// TIA Portal project "PLC_test_DATN" (V16)

(* hardware
DEVICE "S7-1200 station_1"  S7-1200 Station
   slot 0: "Rack_0"  S7-1200 Rack  Rack  V1.0
   slot 1: "PLC_2"  CPU 1214C DC/DC/DC  6ES7 214-1AG40-0XB0  V4.4
*)

// ===== PLC "PLC_2"  CPU 1214C DC/DC/DC =====

VAR_GLOBAL   // PLC tag table "Default tag table"
   "START BUTTON" AT %I0.0 : Bool;
   "SSBELTBEGIN" AT %I0.1 : Bool;
   "SSZ+" AT %I1.3 : Bool;
   "SSZ-" AT %I1.4 : Bool;
   "STOP BUTTON" AT %I1.5 : Bool;
   "GRAB" AT %I1.6 : Bool;
   "LETOUT" AT %I1.7 : Bool;
   "SSX0" AT %I1.0 : Bool;
   "SSX1" AT %I1.1 : Bool;
   "SSX2" AT %I0.4 : Bool;
   "Tag_2" AT %I0.5 : Bool;
   "Tag_3" AT %I0.6 : Bool;
   "SSBELTEND" AT %I0.7 : Bool;
   "SSPUSHERBACK" AT %I0.2 : Bool;
   "SSX3" AT %I1.2 : Bool;
   "SSPUSHERFRONT" AT %I0.3 : Bool;
   "BELTMOTOR" AT %Q0.0 : Bool;
   "HANDPICK" AT %Q0.1 : Bool;
   "HANDLEFT" AT %Q0.3 : Bool;
   "HANDUP" AT %Q0.2 : Bool;
   "PUSHERFRONT" AT %Q0.4 : Bool;
   "HANDRELEASE" AT %Q0.5 : Bool;
   "PUSHERBACK" AT %Q1.1 : Bool;
   "ZPLUS" AT %Q1.2 : Bool;
   "ZMINUS" AT %Q1.3 : Bool;
   "G" AT %Q1.4 : Bool;
   "HANDDOWN" AT %Q0.6 : Bool;
   "HANDRIGHT" AT %Q0.7 : Bool;
   "Tag_12" AT %Q1.0 : Bool;
   "System_Byte" AT %MB2000 : Byte;
   "FirstScan" AT %M2000.0 : Bool;
   "DiagStatusUpdate" AT %M2000.1 : Bool;
   "AlwaysTRUE" AT %M2000.2 : Bool;
   "AlwaysFALSE" AT %M2000.3 : Bool;
   "Clock_Byte" AT %MB5000 : Byte;
   "Clock_10Hz" AT %M5000.0 : Bool;
   "Clock_5Hz" AT %M5000.1 : Bool;
   "Clock_2.5Hz" AT %M5000.2 : Bool;
   "Clock_2Hz" AT %M5000.3 : Bool;
   "Clock_1.25Hz" AT %M5000.4 : Bool;
   "Clock_1Hz" AT %M5000.5 : Bool;
   "Clock_0.625Hz" AT %M5000.6 : Bool;
   "Clock_0.5Hz" AT %M5000.7 : Bool;
   "S0" AT %M1.0 : Bool;
   "S1" AT %M1.1 : Bool;
   "S2" AT %M1.2 : Bool;
   "S3" AT %M1.3 : Bool;
   "S4" AT %M1.4 : Bool;
   "S5" AT %M1.5 : Bool;
   "S6" AT %M1.6 : Bool;
   "S7" AT %M1.7 : Bool;
   "S8" AT %M2.0 : Bool;
   "S9" AT %M2.1 : Bool;
   "S10" AT %M2.2 : Bool;
   "S11" AT %M2.3 : Bool;
   "T00" AT %M2.4 : Bool;
   "T01" AT %M2.5 : Bool;
   "T12" AT %M2.6 : Bool;
   "T23" AT %M2.7 : Bool;
   "T34" AT %M3.0 : Bool;
   "T45" AT %M3.1 : Bool;
   "T56" AT %M3.2 : Bool;
   "T67" AT %M3.3 : Bool;
   "T78" AT %M3.4 : Bool;
   "T89" AT %M3.5 : Bool;
   "T910" AT %M3.6 : Bool;
   "T1011" AT %M3.7 : Bool;
   "T10" AT %M4.0 : Bool;
   "T20" AT %M4.1 : Bool;
   "T30" AT %M4.2 : Bool;
   "T40" AT %M4.3 : Bool;
   "T50" AT %M4.4 : Bool;
   "T60" AT %M4.5 : Bool;
   "T70" AT %M4.6 : Bool;
   "T80" AT %M4.7 : Bool;
   "T90" AT %M5.0 : Bool;
   "T100" AT %M5.1 : Bool;
   "T110" AT %M5.2 : Bool;
   "START" AT %M5.3 : Bool;
   "STOP" AT %M5.4 : Bool;
   "RESET" AT %M5.5 : Bool;
   "PUSHERPOS-" AT %M5.6 : Bool;
   "PUSHERPOS+" AT %M5.7 : Bool;
   "T_1" AT %MD6 : Time;
   "T_2" AT %MD10 : Time;
   "T_3" AT %MD14 : Time;
   "T_4" AT %MD18 : Time;
   "T_5" AT %MD22 : Time;
   "T_6" AT %MD26 : Time;
   "T_7" AT %MD30 : Time;
   "PUSHBACK" AT %M34.0 : Bool;
   "PUSHFRONT" AT %M34.1 : Bool;
   "DOWN" AT %M34.2 : Bool;
   "PICK" AT %M34.3 : Bool;
   "UP" AT %M34.4 : Bool;
   "RELEASE" AT %M34.5 : Bool;
   "RIGHT" AT %M34.6 : Bool;
   "LEFT" AT %M34.7 : Bool;
   "T_8" AT %MD36 : Time;
   "T111" AT %M35.0 : Bool;
   "PULLBACK" AT %M35.1 : Bool;
   "BELT2" AT %M35.2 : Bool;
   "T02" AT %M35.3 : Bool;
   "T03" AT %M35.4 : Bool;
   "T04" AT %M35.5 : Bool;
   "T05" AT %M35.6 : Bool;
   "T06" AT %M35.7 : Bool;
   "T07" AT %M40.0 : Bool;
   "T08" AT %M40.1 : Bool;
   "T09" AT %M40.2 : Bool;
   "T010" AT %M40.3 : Bool;
   "T011" AT %M40.4 : Bool;
   "T410" AT %M40.5 : Bool;
   "T59" AT %M40.6 : Bool;
   "T69" AT %M40.7 : Bool;
   "T79" AT %M41.0 : Bool;
   "T99" AT %M41.1 : Bool;
   "T1010" AT %M41.2 : Bool;
   "T1111" AT %M41.3 : Bool;
   "EMERGENCYSTOP" AT %M41.4 : Bool;
   "AUTOMODE" AT %M41.5 : Bool;
   "MANUALMODE" AT %M41.6 : Bool;
   "RIGHT2" AT %M41.7 : Bool;
   "LEFT2" AT %M42.0 : Bool;
   "DOWN2" AT %M42.1 : Bool;
   "UP2" AT %M42.2 : Bool;
   "PICK2" AT %M42.3 : Bool;
   "RELEASE2" AT %M42.4 : Bool;
   "PUSHBACK2" AT %M42.5 : Bool;
   "PUSHFRONT2" AT %M42.6 : Bool;
   "BELTBEGIN" AT %M42.7 : Bool;
   "BELTEND" AT %M43.0 : Bool;
   "Z+" AT %M43.1 : Bool;
   "Z-" AT %M43.2 : Bool;
   "X0" AT %M43.3 : Bool;
   "X1" AT %M43.4 : Bool;
   "X2" AT %M43.5 : Bool;
   "X3" AT %M43.6 : Bool;
   "AUTO BUTTON" AT %M43.7 : Bool;
   "MANUAL BUTTON" AT %M44.0 : Bool;
   "RESET BUTTON" AT %M44.1 : Bool;
   "BELT" AT %M44.2 : Bool;
   "T74" AT %M44.3 : Bool;
   "T48" AT %M44.4 : Bool;
   "T86" AT %M44.5 : Bool;
   "T91" AT %M44.6 : Bool;
   "X1MODE" AT %M44.7 : Bool;
   "X2MODE" AT %M45.0 : Bool;
   "X3MODE" AT %M45.1 : Bool;
   "T58" AT %M45.2 : Bool;
   "T68" AT %M45.3 : Bool;
   "MEM1" AT %M45.4 : Bool;
   "MEM2" AT %M45.5 : Bool;
   "MEM3" AT %M45.6 : Bool;
   "CAMERA" AT %M45.7 : Bool;
   "TIMEERRORM" AT %M46.0 : Bool;
   "EXTRA" AT %M46.1 : Bool;
END_VAR

DATA_BLOCK "Manual Converter 2_DB"   // DB14
{ S7_Optimized_Access := 'TRUE' }
VERSION : 0.1
// stored: InstanceOfName Manual Converter 2
"Manual Converter 2"
BEGIN
END_DATA_BLOCK

DATA_BLOCK "Auto Converter 2_DB"   // DB19
{ S7_Optimized_Access := 'TRUE' }
VERSION : 0.1
// stored: InstanceOfName Auto Converter 2
"Auto Converter 2"
BEGIN
END_DATA_BLOCK

DATA_BLOCK "Auto SCL 2_DB"   // DB22
{ S7_Optimized_Access := 'TRUE' }
VERSION : 0.1
// stored: InstanceOfName Auto SCL 2
"Auto SCL 2"
BEGIN
END_DATA_BLOCK

DATA_BLOCK "Output Converter 2_DB"   // DB23
{ S7_Optimized_Access := 'TRUE' }
VERSION : 0.1
// stored: InstanceOfName Output Converter 2
"Output Converter 2"
BEGIN
END_DATA_BLOCK

// folder: System blocks/Program resources

DATA_BLOCK "T5"   // DB1
{ S7_Optimized_Access := 'TRUE' }
AUTHOR : Simatic
FAMILY : IEC
NAME : IEC_TMR
VERSION : 1.0
// stored: InstanceOfName IEC_TIMER
"IEC_TIMER"
BEGIN
END_DATA_BLOCK

DATA_BLOCK "T1"   // DB4
{ S7_Optimized_Access := 'TRUE' }
AUTHOR : Simatic
FAMILY : IEC
NAME : IEC_TMR
VERSION : 1.0
// stored: InstanceOfName IEC_TIMER
"IEC_TIMER"
BEGIN
END_DATA_BLOCK

DATA_BLOCK "T2"   // DB5
{ S7_Optimized_Access := 'TRUE' }
AUTHOR : Simatic
FAMILY : IEC
NAME : IEC_TMR
VERSION : 1.0
// stored: InstanceOfName IEC_TIMER
"IEC_TIMER"
BEGIN
END_DATA_BLOCK

DATA_BLOCK "T3"   // DB6
{ S7_Optimized_Access := 'TRUE' }
AUTHOR : Simatic
FAMILY : IEC
NAME : IEC_TMR
VERSION : 1.0
// stored: InstanceOfName IEC_TIMER
"IEC_TIMER"
BEGIN
END_DATA_BLOCK

DATA_BLOCK "T4"   // DB7
{ S7_Optimized_Access := 'TRUE' }
AUTHOR : Simatic
FAMILY : IEC
NAME : IEC_TMR
VERSION : 1.0
// stored: InstanceOfName IEC_TIMER
"IEC_TIMER"
BEGIN
END_DATA_BLOCK

DATA_BLOCK "TP1"   // DB25
{ S7_Optimized_Access := 'TRUE' }
AUTHOR : Simatic
FAMILY : IEC
NAME : IEC_TMR
VERSION : 1.0
// stored: InstanceOfName IEC_TIMER
"IEC_TIMER"
BEGIN
END_DATA_BLOCK

// folder: (top level)

FUNCTION_BLOCK "Manual Converter 2"   // FB5, LAD
{ S7_Optimized_Access := 'TRUE' }
VERSION : 0.1
BEGIN

REGION Network 1
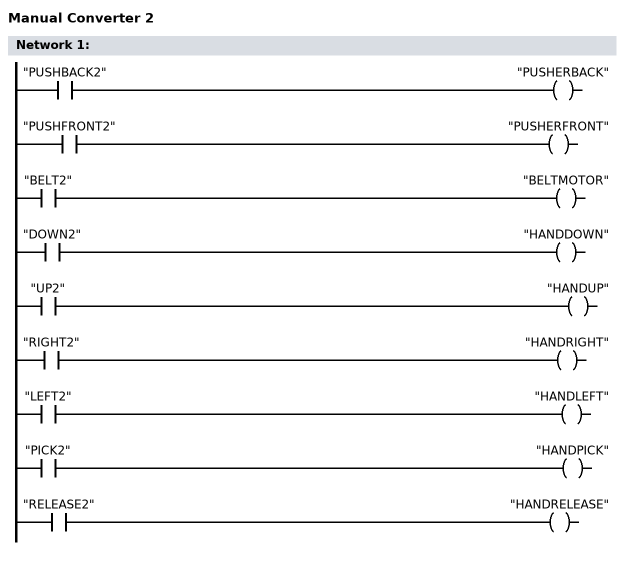
   RUNG wire#powerrail
      Contact( "PUSHBACK2" )
      Coil( "PUSHERBACK" )
   END_RUNG
   RUNG wire#powerrail
      Contact( "PUSHFRONT2" )
      Coil( "PUSHERFRONT" )
   END_RUNG
   RUNG wire#powerrail
      Contact( "BELT2" )
      Coil( "BELTMOTOR" )
   END_RUNG
   RUNG wire#powerrail
      Contact( "DOWN2" )
      Coil( "HANDDOWN" )
   END_RUNG
   RUNG wire#powerrail
      Contact( "UP2" )
      Coil( "HANDUP" )
   END_RUNG
   RUNG wire#powerrail
      Contact( "RIGHT2" )
      Coil( "HANDRIGHT" )
   END_RUNG
   RUNG wire#powerrail
      Contact( "LEFT2" )
      Coil( "HANDLEFT" )
   END_RUNG
   RUNG wire#powerrail
      Contact( "PICK2" )
      Coil( "HANDPICK" )
   END_RUNG
   RUNG wire#powerrail
      Contact( "RELEASE2" )
      Coil( "HANDRELEASE" )
   END_RUNG
   // the same network as SCL:
   "PUSHERBACK" := "PUSHBACK2";
   "PUSHERFRONT" := "PUSHFRONT2";
   "BELTMOTOR" := "BELT2";
   "HANDDOWN" := "DOWN2";
   "HANDUP" := "UP2";
   "HANDRIGHT" := "RIGHT2";
   "HANDLEFT" := "LEFT2";
   "HANDPICK" := "PICK2";
   "HANDRELEASE" := "RELEASE2";
END_REGION
END_FUNCTION_BLOCK

FUNCTION_BLOCK "Auto Converter 2"   // FB6, LAD
{ S7_Optimized_Access := 'TRUE' }
VERSION : 0.1
BEGIN

REGION Network 1
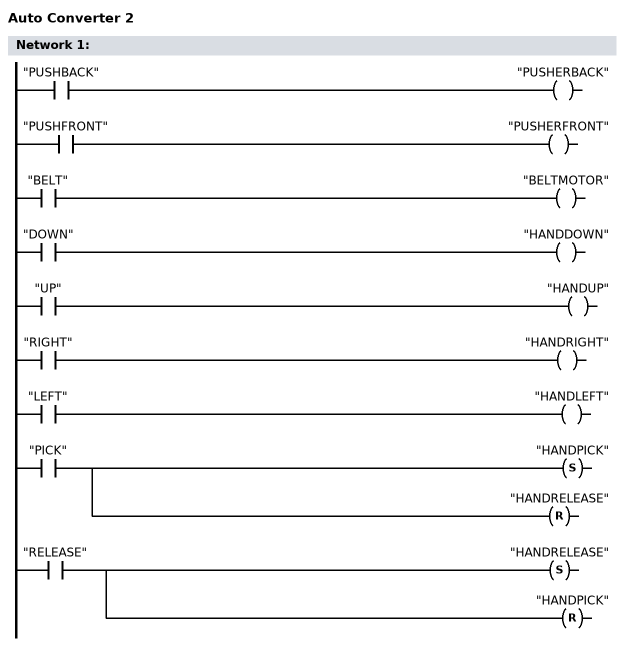
   RUNG wire#powerrail
      Contact( "PUSHBACK" )
      Coil( "PUSHERBACK" )
   END_RUNG
   RUNG wire#powerrail
      Contact( "PUSHFRONT" )
      Coil( "PUSHERFRONT" )
   END_RUNG
   RUNG wire#powerrail
      Contact( "BELT" )
      Coil( "BELTMOTOR" )
   END_RUNG
   RUNG wire#powerrail
      Contact( "DOWN" )
      Coil( "HANDDOWN" )
   END_RUNG
   RUNG wire#powerrail
      Contact( "UP" )
      Coil( "HANDUP" )
   END_RUNG
   RUNG wire#powerrail
      Contact( "RIGHT" )
      Coil( "HANDRIGHT" )
   END_RUNG
   RUNG wire#powerrail
      Contact( "LEFT" )
      Coil( "HANDLEFT" )
   END_RUNG
   RUNG wire#powerrail
      Contact( "PICK" )
      wire#w1
      S_Coil( "HANDPICK" )
   END_RUNG
   RUNG wire#w1
      R_Coil( "HANDRELEASE" )
   END_RUNG
   RUNG wire#powerrail
      Contact( "RELEASE" )
      wire#w2
      S_Coil( "HANDRELEASE" )
   END_RUNG
   RUNG wire#w2
      R_Coil( "HANDPICK" )
   END_RUNG
   // the same network as SCL:
   "PUSHERBACK" := "PUSHBACK";
   "PUSHERFRONT" := "PUSHFRONT";
   "BELTMOTOR" := "BELT";
   "HANDDOWN" := "DOWN";
   "HANDUP" := "UP";
   "HANDRIGHT" := "RIGHT";
   "HANDLEFT" := "LEFT";
   IF "PICK" THEN
       "HANDPICK" := TRUE;
       "HANDRELEASE" := FALSE;
   END_IF;
   IF "RELEASE" THEN
       "HANDRELEASE" := TRUE;
       "HANDPICK" := FALSE;
   END_IF;
END_REGION
END_FUNCTION_BLOCK

FUNCTION_BLOCK "Output Converter 2"   // FB7, LAD
{ S7_Optimized_Access := 'TRUE' }
VERSION : 0.1
BEGIN

REGION Network 1
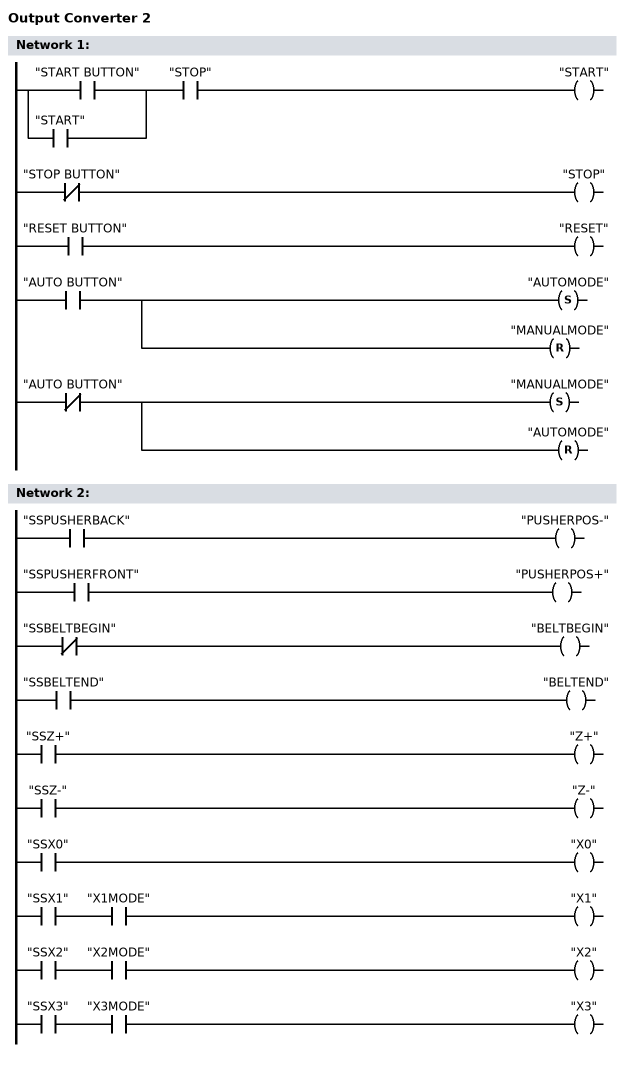
   RUNG wire#powerrail
      Contact( "START BUTTON" )
      wire#w1
      Contact( "STOP" )
      Coil( "START" )
   END_RUNG
   RUNG wire#powerrail
      Contact( "START" )
   END_RUNG wire#w1
   RUNG wire#powerrail
      I_Contact( "STOP BUTTON" )
      Coil( "STOP" )
   END_RUNG
   RUNG wire#powerrail
      Contact( "RESET BUTTON" )
      Coil( "RESET" )
   END_RUNG
   RUNG wire#powerrail
      Contact( "AUTO BUTTON" )
      wire#w2
      S_Coil( "AUTOMODE" )
   END_RUNG
   RUNG wire#w2
      R_Coil( "MANUALMODE" )
   END_RUNG
   RUNG wire#powerrail
      I_Contact( "AUTO BUTTON" )
      wire#w3
      S_Coil( "MANUALMODE" )
   END_RUNG
   RUNG wire#w3
      R_Coil( "AUTOMODE" )
   END_RUNG
   // the same network as SCL:
   "START" := ("START BUTTON" OR "START") AND "STOP";
   "STOP" := NOT "STOP BUTTON";
   "RESET" := "RESET BUTTON";
   IF "AUTO BUTTON" THEN
       "AUTOMODE" := TRUE;
       "MANUALMODE" := FALSE;
   END_IF;
   IF NOT "AUTO BUTTON" THEN
       "MANUALMODE" := TRUE;
       "AUTOMODE" := FALSE;
   END_IF;
END_REGION

REGION Network 2
   RUNG wire#powerrail
      Contact( "SSPUSHERBACK" )
      Coil( "PUSHERPOS-" )
   END_RUNG
   RUNG wire#powerrail
      Contact( "SSPUSHERFRONT" )
      Coil( "PUSHERPOS+" )
   END_RUNG
   RUNG wire#powerrail
      I_Contact( "SSBELTBEGIN" )
      Coil( "BELTBEGIN" )
   END_RUNG
   RUNG wire#powerrail
      Contact( "SSBELTEND" )
      Coil( "BELTEND" )
   END_RUNG
   RUNG wire#powerrail
      Contact( "SSZ+" )
      Coil( "Z+" )
   END_RUNG
   RUNG wire#powerrail
      Contact( "SSZ-" )
      Coil( "Z-" )
   END_RUNG
   RUNG wire#powerrail
      Contact( "SSX0" )
      Coil( "X0" )
   END_RUNG
   RUNG wire#powerrail
      Contact( "SSX1" )
      Contact( "X1MODE" )
      Coil( "X1" )
   END_RUNG
   RUNG wire#powerrail
      Contact( "SSX2" )
      Contact( "X2MODE" )
      Coil( "X2" )
   END_RUNG
   RUNG wire#powerrail
      Contact( "SSX3" )
      Contact( "X3MODE" )
      Coil( "X3" )
   END_RUNG
   // the same network as SCL:
   "PUSHERPOS-" := "SSPUSHERBACK";
   "PUSHERPOS+" := "SSPUSHERFRONT";
   "BELTBEGIN" := NOT "SSBELTBEGIN";
   "BELTEND" := "SSBELTEND";
   "Z+" := "SSZ+";
   "Z-" := "SSZ-";
   "X0" := "SSX0";
   "X1" := "SSX1" AND "X1MODE";
   "X2" := "SSX2" AND "X2MODE";
   "X3" := "SSX3" AND "X3MODE";
END_REGION
END_FUNCTION_BLOCK

FUNCTION_BLOCK "Auto SCL 2"   // FB8, SCL
{ S7_Optimized_Access := 'TRUE' }
VERSION : 0.1
BEGIN
   "T1".TON(IN := "S5",
            PT := T#2S);

   "T2".TON(IN := "S9",
            PT := T#2S);


   "T3".TON(IN := "S7",
            PT := T#1S,
            Q => "MEM1");

   "T5".TON(IN:="S4",
            PT:=T#1S);


   "TP1".TP(IN := "MEM1" AND NOT "MEM2",
            PT := T#50MS,
            Q => "MEM3");

   "T4".TON(IN := "MEM1" AND NOT "MEM2" AND NOT "MEM3",
            PT := T#250MS,
            Q => "MEM2");

   //TRANSITION EQUATION

   "T00" := "FirstScan";
   "T01" := "S0" AND "START";
   "T12" := "S1" AND "PUSHERPOS-" AND "BELTBEGIN" AND "START";
   "T23" := "S2" AND "PUSHERPOS+" AND "START";
   "T34" := "S3" AND "BELTEND" AND "START";
   "T45" := "S4" AND "Z-" AND "START";
   "T56" := "S5" AND "T1".Q AND "START";
   "T67" := "S6" AND "Z+" AND "START";
   "T78" := "S7" AND ("X1" OR "X2" OR "X3") AND "START";
   "T89" := "S8" AND (("Z-" AND "START") OR "RESET");
   "T910" := "S9" AND (("T2".Q AND "START") OR "RESET");
   "T1011" := "S10" AND (("Z+" AND "START") OR "RESET");
   "T111" := "S11" AND "X0" AND "START";


   "T10" := "S1" AND (NOT "START" AND "RESET");
   "T20" := "S2" AND (NOT "START" AND "RESET");
   "T30" := "S3" AND (NOT "START" AND "RESET");

   "T110" := "S11" AND (NOT "START" AND "RESET");

   "T410" := "S4" AND NOT "START" AND "RESET";
   "T59" := "S5" AND NOT "START" AND "RESET";
   "T69" := "S6" AND NOT "START" AND "RESET";
   "T79" := "S7" AND NOT "START" AND "RESET";




   //STATE EQUATION
   "S0" := ("S0" OR "T00" OR "T10" OR "T20" OR "T30" OR "T40" OR "T50" OR "T60" OR "T70" OR "T80" OR "T90" OR "T100" OR "T110") AND NOT "T01";
   "S1" := ("S1" OR "T01" OR "T111") AND NOT "T10" AND NOT "T12";
   "S2" := ("S2" OR "T12") AND NOT "T20" AND NOT "T23";
   "S3" := ("S3" OR "T23") AND NOT "T30" AND NOT "T34";
   "S4" := ("S4" OR "T34") AND NOT "T40" AND NOT "T45" AND NOT "T410";
   "S5" := ("S5" OR "T45") AND NOT "T50" AND NOT "T56" AND NOT "T59";
   "S6" := ("S6" OR "T56") AND NOT "T60" AND NOT "T67" AND NOT "T69";
   "S7" := ("S7" OR "T67") AND NOT "T70" AND NOT "T78" AND NOT "T79";
   "S8" := ("S8" OR "T78") AND NOT "T80" AND NOT "T89";
   "S9" := ("S9" OR "T89" OR "T59" OR "T69" OR "T79") AND NOT "T90" AND NOT "T910";
   "S10" := ("S10" OR "T910" OR "T410") AND NOT "T100" AND NOT "T1011";
   "S11" := ("S11" OR "T1011") AND NOT "T110" AND NOT "T111";

   //OUTPUT EQUATION
   "PUSHBACK" := "S1" AND "START";
   "PUSHFRONT" := "S0" OR ("S2" AND "START");
   "BELT" := "S3" AND "START" AND NOT "CAMERA";
   "DOWN" := ("S4" AND "T5".Q) OR "S8";
   "PICK" := "S5";
   "UP" := "S0" OR "S6" OR "S10";
   "RIGHT" := ("S7" AND NOT "MEM1") OR "MEM3" ;
   "RELEASE" :="S9";
   "LEFT" := "S0" OR "S11";
END_FUNCTION_BLOCK

FUNCTION "MHJ-PLC-Lab-Function-S71200" : Void   // FC9000, SCL
{ S7_Optimized_Access := 'TRUE' }
VERSION : 0.1
   VAR_TEMP
      rdTimeReturn : Int;
      outputTime : DTL;
      SyncVal : Byte;
      forVal : Int;
      forVal_2 : Int;
      Value : Byte;
   END_VAR
   VAR CONSTANT
      CompVal : Byte := 16#34;
      Value_01 : Byte := 16#11;
      Value_01_DW : DWord := 16#A165_D992;
      Value_02_DW : DWord := 16#58BE_4401;
   END_VAR
BEGIN

   #Value:=PEEK(area := 16#82,
        dbNumber := 0,
        byteOffset := 511);
   #Value := #Value + 1;

   POKE(area := 16#82,
        dbNumber := 0,
        byteOffset := 511,
        value := #Value);

   POKE(area:=16#81,
        dbNumber:=0,
        byteOffset:=1016,
        value:=#Value_01_DW);

   POKE(area := 16#81,
        dbNumber := 0,
        byteOffset := 1020,
        value := #Value_02_DW);

   POKE(area := 16#81,
        dbNumber := 0,
        byteOffset := 511,
        value := B#16#00);

   FOR #forVal := 0 TO 120 DO
       FOR #forVal_2:=0 TO 10 DO
           #rdTimeReturn:=RD_SYS_T(#outputTime);
           #rdTimeReturn := WR_SYS_T(#outputTime);
           #rdTimeReturn := RD_SYS_T(#outputTime);
           #rdTimeReturn := WR_SYS_T(#outputTime);
       END_FOR;
       #SyncVal:= PEEK(area := 16#81,
                      dbNumber := 0,
                      byteOffset := 511);
       IF #SyncVal = #CompVal THEN
          GOTO M_1;
       END_IF;
   END_FOR;
   RETURN;

   M_1:
   POKE(area := 16#81,
        dbNumber := 0,
        byteOffset := 511,
        value := B#16#0);
END_FUNCTION

ORGANIZATION_BLOCK "Main"   // OB1, LAD, ProgramCycle
TITLE = "Main Program Sweep (Cycle)"
{ S7_Optimized_Access := 'TRUE' }
VERSION : 0.1
   VAR_INPUT
      Initial_Call : Bool;   // Initial call of this OB
      Remanence : Bool;   // =True, if remanent data are available
   END_VAR
BEGIN

REGION Network 1
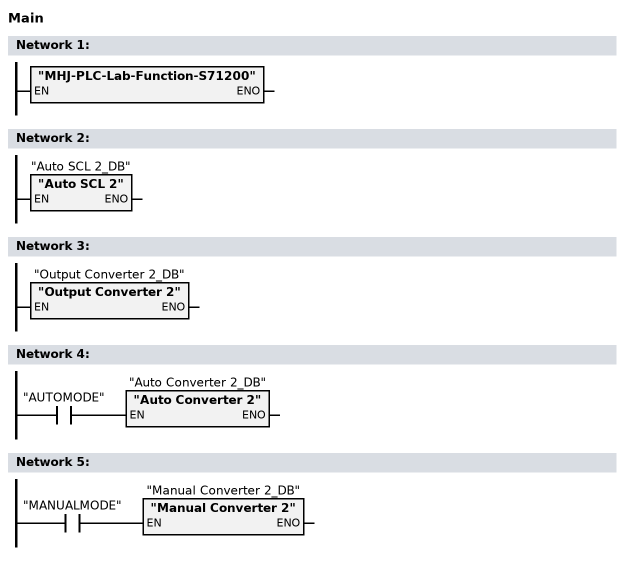
   RUNG wire#powerrail
      "MHJ-PLC-Lab-Function-S71200"()
   END_RUNG
   // the same network as SCL:
   "MHJ-PLC-Lab-Function-S71200"();
END_REGION

REGION Network 2
   RUNG wire#powerrail
      "Auto SCL 2_DB"()
   END_RUNG
   // the same network as SCL:
   "Auto SCL 2_DB"();   // "Auto SCL 2"
END_REGION

REGION Network 3
   RUNG wire#powerrail
      "Output Converter 2_DB"()
   END_RUNG
   // the same network as SCL:
   "Output Converter 2_DB"();   // "Output Converter 2"
END_REGION

REGION Network 4
   RUNG wire#powerrail
      Contact( "AUTOMODE" )
      "Auto Converter 2_DB"()
   END_RUNG
   // the same network as SCL:
   IF "AUTOMODE" THEN
       "Auto Converter 2_DB"();   // "Auto Converter 2"
   END_IF;
END_REGION

REGION Network 5
   RUNG wire#powerrail
      Contact( "MANUALMODE" )
      "Manual Converter 2_DB"()
   END_RUNG
   // the same network as SCL:
   IF "MANUALMODE" THEN
       "Manual Converter 2_DB"();   // "Manual Converter 2"
   END_IF;
END_REGION
END_ORGANIZATION_BLOCK